{attribute 'hide_all_locals'}
FUNCTION_BLOCK EnableGroup IMPLEMENTS ITask
VAR_INPUT
END_VAR
VAR_OUTPUT
END_VAR
VAR
	groupEnable			: MC_GroupEnable;
	_caGroup			: ICollisionGroup;
	State: INT;
	_enableGroup : BOOL;
	_busy : BOOL;
	_error : BOOL;
	_done : BOOL;
	Logger : TcMessage_Ext;
END_VAR

CASE State OF
	0:
		IF _enableGroup THEN
			_done := FALSE;
			_error := FALSE;
			_busy := TRUE;
			groupEnable.Execute := TRUE;
			IF groupEnable.Busy THEN
				State := 10;
				_enableGroup := FALSE;
				logger.Send(TC_EVENTS.XtsCAGroupEvents.CAGroupEnabling,'');
			END_IF
		END_IF
	
	10:
		IF NOT groupEnable.Busy THEN
			IF groupEnable.Done THEN
				_done := TRUE;
				logger.Send(TC_EVENTS.XtsCAGroupEvents.CAGroupEnabled,'');
			ELSIF groupEnable.Error THEN
				_error := TRUE;
				logger.Send(TC_EVENTS.XtsCAGroupEvents.CAGroupEnableError,'');
			END_IF
			_busy := FALSE;
			groupEnable.Execute := false;
			State := 0;
		END_IF
END_CASE


groupEnable(AxesGroup := _caGroup.GroupRef);

METHOD Abort : BOOL
groupEnable.Execute := FALSE;
Abort := TRUE;
State := 0;
END_METHOD

PROPERTY Busy : BOOL
GET
Busy := _busy;
END_GET
END_PROPERTY

PROPERTY Done : BOOL
GET
Done := _done;
END_GET
END_PROPERTY

PROPERTY Error : BOOL
GET
Error := _error;
END_GET
END_PROPERTY

METHOD Execute : BOOL
Execute := _enableGroup := true;
END_METHOD

METHOD FB_init : BOOL
VAR_INPUT
	bInitRetains : BOOL; // if TRUE, the retain variables are initialized (warm start / cold start)
	bInCopyCode : BOOL;  // if TRUE, the instance afterwards gets moved into the copy code (online change)
	CAGroup : ICollisionGroup;	
END_VAR
_caGroup := CAGroup;
END_METHOD

END_FUNCTION_BLOCK

(* stored: Version 1.1.0.1, ProductVersion 3.1.4024.11
   POU EnableGroup: Id {78c0ffeb-f751-4064-9ca5-f5352de8dccc}, SpecialFunc None
   Method Abort: Id {b71dbe64-bf42-4f8d-bc93-a820b314190e}
   Property Busy: Id {844fe327-b432-4d9b-9ff8-674b403712de}
   Get Get: Id {9de7276e-68b8-471b-acbe-4af805d8f9d4}
   Property Done: Id {96fe3f04-3684-47c6-96b8-040adc9ccb95}
   Get Get: Id {752b21aa-907b-4aba-b185-74a8d165978c}
   Property Error: Id {91a57102-e8a8-46ee-bdd6-0ba18161e2fa}
   Get Get: Id {f8961f71-0d32-45d5-9893-2036d33f4a14}
   Method Execute: Id {46988e83-7049-4ed9-931d-ac6221516616}
   Method FB_init: Id {b5caa772-6afb-4d2b-9da8-e7bb1ea9e9b8} *)
